{attribute 'TcGenerated'}
{attribute 'no-analysis'}
{attribute 'linkalways'}
// This function has been automatically generated from the project information.
VAR_GLOBAL CONSTANT
	{attribute 'const_non_replaced'}
	stLibVersion_TwinCat_Dynamic_Collections : ST_LibVersion := (iMajor := 1, iMinor := 0, iBuild := 9, iRevision := 0, nFlags := 0, sVersion := '1.0.9');
END_VAR

(* stored: Version 1.1.0.1
   GVL Global_Version: Id {1cd6a6bf-c905-4a98-83a0-71aa67a98824} *)
